INTERFACE iTwoDirectionalMotorWithFast EXTENDS iTwoDirectionalMotor // Two directional motor with run fast commands

METHOD CmdRunCCWFast : BOOL
VAR_INPUT
END_VAR
END_METHOD

METHOD CmdRunCWFast : BOOL
VAR_INPUT
END_VAR
END_METHOD

END_INTERFACE

(* stored: Version 1.1.0.1, ProductVersion 3.1.4024.10
   Itf iTwoDirectionalMotorWithFast: Id {992056b8-17e9-00b5-0fc7-3c5cd8787b1d}
   Method CmdRunCCWFast: Id {32b655a9-8667-0ca6-06ce-b62af57655e2}
   Method CmdRunCWFast: Id {d70282e7-67d5-0030-1a17-e8ea495802ef} *)
